# EPICS substitutions: examplesTop/ndsex1App/Db/Firmware.substitutions
file "nds3_Firmware.template" {
pattern
{
    BOARDTYPE,
    BOARDTYPEIDX,
    CBS1,
    CBS2,
    STATEMACHINE_PARENT,
    STATEMACHINE_NAME,
    FIRMWARE_NAME,
}

{
    "B",
    "0",
    "TEST",
    "FCT0",
    "Firm-",
    "StateMachine"
    "Firm",
}

}
